// TIA Portal V21 export
DATA_BLOCK "REVAMP"   // DB1
{ S7_Optimized_Access := 'FALSE' }
   VAR
      L1 : String[80] := '$L$R                       CLIENT:- M/s. KWALITY PHARMACEUTICALS LTD             ';
      L2 : String[80] := '$L$R 6TH MILE STONE, VILL.NAG KALAN, MAJITHA ROAD, AMRITSAR, PUNJAB-143601';
      L3 : String[80] := '$L$R                                    BATCH DATA';
      L4 : String[80] := '$L$R                                STEAM STERILIZER   ';
      L5 : String[80] := '$L$R             -----------------------------------------------------';
      L6 : String[80] := '$L$REQUIPMENT ID        :';
      L7 : String[80] := '$L$RPRODUCT NAME        :';
      L8 : String[80] := '$L$RBATCH NO            :';
      L9 : String[80] := '                                                             DATE: 04/05/2025';
      L10 : String[80] := '  PROCESS STARTED AT  :13:09:19';
      L11 : String[80] := '$L$ROPERATOR NAME       :';
      L12 : String[80] := '$L$RPROCESS                    :    ';
      L13 : String[80] := '$L$R        :';
      L14 : String[80] := '-------------';
      L15 : String[80] := '$L$R   ';
      L16 : String[80] := '$L$R                           CYCLE COMPLETED   ';
      L17 : String[80] := '$L$R                 ';
      L18 : String[80] := '$L$R                                          ';
      L19 : String[80] := '$L$R DONE BY  :                                 CHECKED BY :';
      L20 : String[80] := '$L$R******************************************************************************';
      L21 : String[80] := '$L$R DATE  :                                     DATE :';
      L22 : String[80] := '$L$R  SUMMARY OF VACUUM LEAK TEST  ';
      L23 : String[80] := '$L$R******************************************************************************';
      L24 : String[80] := '$L$R  TIME  : PRESSURE:  CH-1  :  CH-2  :  CH-3  :  CH-4  :  CH-5  :  STATUS      ';
      L25 : String[90] := '$L$R           :  DZ    :  MHZ   :  ST IN :  ST OUT:  CZ UP :  CZDOWN:  SPEED ';
      L26 : String[80] := '$L$R        :  BAR    :  DEG.C :  DEG.C :  DEG.C :  DEG.C :  DEG.C :   ';
      L27 : String[80] := '$L$R------------------------------------------------------------------------------';
      L28 : String[80] := '  13:09:20    1.032    116.2    120.6    119.9    119.4    120.2 HEATUP-1 HOLD';
      L29 : String[80] := '$L$R                                                                   ';
      L30 : String[80] := '$L$R------------------------------------------------------------------------------';
      L31 : String[80] := '               RECEIPE TYPE :                                                   ';
      L32 : String[80] := '--------------------------------------------------------------------------------';
      ALM1 : String[80] := '$L$R13  9 20';
      ALM2 : String[80] := '$L$R13  9 20';
      ALM3 : String[80] := '$L$R13  9 20';
      ALM4 : String[80] := '$L$R13  9 20';
      ALM5 : String[80] := '$L$R13  9 20';
      ALM6 : String[80] := '$L$R13  9 20';
      ALM7 : String[80] := '$L$R13  9 20';
      ALM8 : String[80] := '$L$R13  9 20';
      ALM9 : String[80] := '$L$R13  9 20';
      ALM10 : String[80] := '$L$R13  9 20';
      ALM11 : String[80] := '$L$R13  9 20';
      ALM12 : String[80] := '$L$R13  9 20';
      ALM13 : String[80] := '$L$R13  9 20';
      ALM14 : String[80] := '$L$R13  9 20';
      ALM15 : String[80] := '$L$R13  9 20';
      ALM16 : String[80] := '$L$R13  9 20';
      ALM17 : String[80] := '$L$R13  9 20';
      ALM18 : String[80] := '$L$R13  9 20';
      ALM19 : String[80] := '$L$R13  9 20';
      ALM20 : String[80] := '$L$R13  9 20';
      ALM21 : String[80] := '$L$RCHECKED BY              :                   VERIFIED BY               :';
      "BATCH SIZE" : String[80] := '  CYCLE NO            :';
      "CONTAINER SIZE" : String[80] := '  CONTAINER SIZE      :';
      "BLANK LINE" : String[80] := '                                                                ';
      ALM22 : String[80] := '    :  :       STABILIZING ZONE PRESSURE LOW/PLEASE CHECK GAUGE OR BLOWER ';
      zero : String[80] := '0';
      pv : String[80] := '';
      COLAN : String[80] := ':';
      T1 : String[80] := '13:';
      T2 : String[80] := '13:09';
      T3 : String[80] := '13:09:';
      T4 : String[80] := '13:09:20';
      T5 : String[80] := '';
      HOURS_P : String[80] := '13';
      MIN_P : String[80] := ' 9';
      SEC_P : String[80] := '20';
      HOURS_P_1 : String[80] := '13';
      MIN_P_1 : String[80] := '09';
      SEC_P_1 : String[80] := '20';
      CH1 : String[80] := ' 1.032';
      CH2 : String[80] := '116.2';
      CH3 : String[80] := '120.6';
      CH4 : String[80] := '119.9';
      CH5 : String[80] := '119.4';
      CH6 : String[80] := '120.2';
      CONVEYOR : String[80] := 'HEATUP-1 HOLD';
      SPACE_1 : String[80] := ' ';
      SPACE_2 : String[80] := '  ';
      SPACE_3 : String[80] := '   ';
      SPACE_4 : String[80] := '    ';
      C1 : String[80] := '  13:09:20    1.032    116.2    120.6    119.9    119.4    120.2 ';
      C2 : String[80] := '';
      C3 : String[80] := '';
      L10_2 : String[80] := '  PROCESS STARTED AT  :';
      L9_2 : String[80] := '                                                             DATE: ';
      DATE_P : String[80] := ' 4';
      MONTH_P : String[80] := ' 5';
      YEAR_P : String[80] := '2025';
      DATE_P_1 : String[80] := '04';
      MONTH_P_1 : String[80] := '05';
      YEAR_P_1 : String[80] := '2025';
      SLASH : String[80] := '/';
      "DATE CONCATE" : String[80] := '04/05/2025';
      ALM_P_1 : String[80] := '    EMERGENCY PRESSED ';
      ALM_P_2 : String[80] := '    TURBINE VFD TRIP ';
      ALM_P_3 : String[80] := '    CONVEYOR SUPPLY FAIL ';
      ALM_P_4 : String[80] := '     LAF SUPLY FAIL ';
      ALM_P_5 : String[80] := '    TURBINE SUPLY FAIL';
      ALM_P_6 : String[80] := '    VAPOR EXHAUST SUPLY FAIL';
      ALM_P_7 : String[80] := '    HEATER SUPLY FAIL';
      ALM_P_8 : String[80] := '    TEMPERATURE OVERSHOOT';
      ALM_P_9 : String[80] := '    VAPOUR EXHAUST TRIP';
      ALM_P_10 : String[80] := '    PHASE FAIL ';
      ALM_P_11 : String[80] := '    DRYING ZONE PRESSURE LOW/PLEASE CHECK GAUGE OR BLOWER ';
      ALM_P_12 : String[80] := '    COOLING ZONE PRESSURE LOW/PLEASE CHECK GAUGE OR BLOWER ';
      ALM_P_13 : String[80] := '    STERILIZING ZONE PREESURE LOW/PLEASE CHECK GAUGE OR TURBINE ';
      ALM_P_14 : String[80] := '    CONVEYOR VFD OVERLOAD ';
      ALM_P_15 : String[80] := '    MAIN HEAT RTD SENSOR FAIL ';
      ALM_P_16 : String[80] := '    STERILE IN RTD SENSOR FAIL ';
      ALM_P_17 : String[80] := '    STERILE OUT RTD SENSOR FAIL ';
      ALM_P_18 : String[80] := '    DROP IN STERLIZATION ZONE TEMPERATURE ';
      ALM_P_19 : String[80] := '    SHUTDOWN CYCLE STARTED ';
      ALM_P_20 : String[80] := '    *****PROCESS COMPLETED*****';
      ALM_P_22 : String[80] := '    STABILIZING ZONE PRESSURE LOW/PLEASE CHECK GAUGE OR BLOWER ';
      ADD2 : String[80] := '$L$R                  AMRITSAR-143001. P';
      "CYCLE STOP" : String[80] := '   ******CYCLE ABORTED****** ';
   END_VAR
BEGIN
END_DATA_BLOCK
